Fanuc TP program (LS listing): CONDIO.LS

/PROG  CONDIO
/ATTR
OWNER		= MNEDITOR;
COMMENT		= "CondIo";
PROG_SIZE	= 0;
CREATE		= DATE 26-01-01  TIME 00:00:00;
MODIFIED	= DATE 26-01-01  TIME 00:00:00;
FILE_NAME	= ;
VERSION		= 0;
LINE_COUNT	= 4;
MEMORY_SIZE	= 0;
PROTECT		= READ_WRITE;
TCD:  STACK_SIZE	= 0,
      TASK_PRIORITY	= 50,
      TIME_SLICE	= 0,
      BUSY_LAMP_OFF	= 0,
      ABORT_REQUEST	= 0,
      PAUSE_REQUEST	= 0;
DEFAULT_GROUP	= 1,*,*,*,*;
CONTROL_CODE	= 00000000 00000000;
/MN
   1:  !RAPID CondProbe.CondIo ;
   2:  IF (GI[1]=0 AND DI[1]=OFF) THEN ;
   3:  R[6:nIo]=R[6:nIo]+1    ;
   4:  ENDIF ;
/POS
/END
